TYPE T_Ctrl_SIf_JCL_Par :
STRUCT
END_STRUCT
END_TYPE

(* stored: Version 1.1.0.1, ProductVersion 3.1.0.26
   DUT T_Ctrl_SIf_JCL_Par: Id {42e642f6-1cfb-402c-9eda-1469d678ed20} *)
